(* PLC project Aufgabe2SPS, Beckhoff Automation GmbH TwinCAT PLC Control 3.5.13.20 *)
(* stored: creationDateTime 2020-03-24T21:12:55.1576625, modificationDateTime 2020-03-24T21:12:55.1616657 *)

TYPE ST_STATUS_WORD_DATA :
STRUCT
	inLenght : INT;
   overrunError  :  BOOL;
   framingError  :  BOOL;
   parityError  :  BOOL;
   bufferFull  :  BOOL;
   initAccepted  :  BOOL;
   receiveRequest  :  BOOL;
   transmitAccepted  :  BOOL;		

END_STRUCT
END_TYPE

FUNCTION_BLOCK FB_EdgeDetector
VAR_INPUT
	b_InputSignal_k : BOOL;
END_VAR
VAR_OUTPUT
	b_PositiveEdge : BOOL;
	b_NegativeEdge : BOOL;
END_VAR
VAR
	b_InputSignal_k_1 : BOOL;
END_VAR

                  b_PositiveEdge := b_InputSignal_k AND NOT b_InputSignal_k_1;
b_NegativeEdge := NOT b_InputSignal_k AND b_InputSignal_k_1;

b_InputSignal_k_1 := b_InputSignal_k;
                
END_FUNCTION_BLOCK

FUNCTION F_AdditionFunction : INT
VAR_INPUT
	i_var1 : INT;
	i_var2 : INT;
END_VAR
VAR
	
END_VAR

                  F_AdditionFunction := i_var1 + i_var2;
                
END_FUNCTION

FUNCTION F_DivisionFunction : INT
VAR_INPUT
	i_var1 : INT;
	i_var2 : INT;
END_VAR
VAR
	
END_VAR

                  IF i_var2 = 0 THEN
	F_DivisionFunction := 0;
ELSE	
	F_DivisionFunction := i_var1 / i_var2;
END_IF

                
END_FUNCTION

FUNCTION F_STATUS_WORD_PROC : ST_STATUS_WORD_DATA
VAR_INPUT
	w_StatusWord : WORD;
END_VAR
VAR
END_VAR

                  

F_STATUS_WORD_PROC.transmitAccepted := w_StatusWord.0;
F_STATUS_WORD_PROC.parityError := w_StatusWord.1;
F_STATUS_WORD_PROC.initAccepted := w_StatusWord.2;
F_STATUS_WORD_PROC.bufferFull := w_StatusWord.3;
F_STATUS_WORD_PROC.parityError := w_StatusWord.4;
F_STATUS_WORD_PROC.framingError := w_StatusWord.5;
F_STATUS_WORD_PROC.overrunError := w_StatusWord.6;
F_STATUS_WORD_PROC.inLenght := WORD_TO_INT(SHR(w_StatusWord,8));
                
END_FUNCTION

PROGRAM MAIN
VAR
	// Lokale Variablen um die Funktionen
	// F_AdditionFunction und F_DivisionFunction zu testen
	i_var1   : INT;
	i_var2   : INT;
	i_addRes : INT;
	i_divRes : INT;
	
	// 16 bits
	w_myword : WORD := 16#5D7A;
	w_divRes : WORD;
	
	// 32 bits
	dw_mydword : DWORD;
	dw_mydword1 : DWORD;
	
	w_testWord : WORD;
	
	st_resRsProt : ST_STATUS_WORD_DATA;
	
	// Array von REAL, Dimension 10
	// arr_r_testArray : ARRAY[0..9] OF REAL;
	arr_r_testArray : ARRAY[1..10] OF REAL;
	
	// Variablen für FOR Schleife
	r_SummeArray : REAL;
	r_MulArray : REAL;
	
	// Variabel für FOR Schleife
	i_SchleifeIterVar : INT;
	
	// Edge detektor 2 Mal instanzieren
	fbEdgeDetectorGelb : FB_EdgeDetector;
	fbEdgeDetectorBlau : FB_EdgeDetector;
	
	// "Software" Taster um Edge Detektor zu testen
	bGelbTaster : BOOL;
	bBlauTaster : BOOL;
	
	// TRUE if positive Flanke bei gelbem Taster
	bGelbPositivEdge : BOOL;
	
	
END_VAR

                  // Aufruf Funktionen Addition/Division direkt vom Main
i_addRes := F_AdditionFunction(i_var1, i_var2);
i_divRes := F_DivisionFunction(i_var1, i_var2);

// Aufruf Funktionen Addition/Division direkt vom DoSomeMath
P_DoSomeMath.i_var1 := i_var1;
P_DoSomeMath.i_var2 := i_var2;
P_DoSomeMath();
i_addRes := P_DoSomeMath.i_addRes;
i_divRes := P_DoSomeMath.i_divRes;

// Teilung durch 8 -> shift right 3 bits
w_divRes := SHR(w_myword, 3);

// Multiplikation mit 8 -> shift left 3 bits
dw_mydword := SHL(w_myword, 3);

// Vier höchsten bits auf 1 setzen 
dw_mydword1 := dw_mydword OR 16#F0000000;

// Aufruf Funktion für RS232 Protokoll
// Auswertung vom Statuswort
st_resRsProt := F_STATUS_WORD_PROC(w_testWord);
 
// FOR Schleife um die Elemente von Array zusammen zu addieren
// bzw. zu multiplizieren
r_SummeArray := 0.0;
r_MulArray   := 1.0;
FOR i_SchleifeIterVar := 1 TO 10 DO
	r_SummeArray := r_SummeArray + arr_r_testArray[i_SchleifeIterVar];
	r_MulArray := r_MulArray * arr_r_testArray[i_SchleifeIterVar];
END_FOR


fbEdgeDetectorGelb(b_InputSignal_k := bGelbTaster);
bGelbPositivEdge := fbEdgeDetectorGelb.b_PositiveEdge;
// Alternativ, Funktionsausruf + Zuweisung Ergebnis in einem Schritt
// fbEdgeDetectorGelb(b_InputSignal_k := bGelbTaster, b_PositiveEdge => bGelbPositivEdge);
IF bGelbpositivEdge THEN
	// Hier Brekpoint setzen mit F9 um EdgeDetector zu testen
	r_MulArray := 0;
END_IF
 
fbEdgeDetectorBlau(b_InputSignal_k := bBlauTaster);
                
END_PROGRAM

PROGRAM P_DoSomeMath
VAR
END_VAR
// VAR_INPUT und VAR_OUTPUT müssen vor Hand
// hinzugefügt werden!!
VAR_INPUT
	i_var1 : INT;
	i_var2 : INT;
END_VAR
VAR_OUTPUT
	i_addRes : INT;
	i_divRes : INT;
END_VAR

                  
                
END_PROGRAM

CONFIGURATION Application
  RESOURCE Aufgabe2SPS ON PLC
    TASK PlcTask(INTERVAL := T#0ms, PRIORITY := 20);
    PROGRAM MAIN WITH PlcTask : MAIN;
  END_RESOURCE
END_CONFIGURATION
